(* CoDeSys 2.3 export: TECHMODULE_KINEMATICS.EXP *)
(* Libraries: 03_ApplicationModules\MPLCAxisGroupControl_Kinematics.lib 30.1.17 00:00:00, 03_ApplicationModules\MPLCAxisGroupControl_Kinematics_Internal_Inst1.lib 30.1.17 00:00:00, 04_InterpolatedMotion\MPLCKinematics.lib 30.1.17 00:00:00, 04_InterpolatedMotion\MPLCKinematics_UserKin.lib 30.1.17 00:00:00, 04_InterpolatedMotion\MPLCKinematics_UserLookAhead.lib 30.1.17 00:00:00, 04_InterpolatedMotion\MPLCSimu3D.lib 30.1.17 00:00:00, 11_System\SysLibStr.lib 27.1.17 13:50:06, Internal\MPLCIntern_Kinematics.lib 30.1.17 00:00:00, Internal\MPLCIntern_Kinematics_BC.lib 30.1.17 00:00:00, Internal\MPLCIntern_Kinematics_Small.lib 30.1.17 00:00:00 *)

(* Global variable list: AxisGroupControl_Kinematics/Examples/GlobalVar_AxisGroupControl_Kinematics_Examples *)
VAR_GLOBAL
	(* !!! Do not remove '{flag extrasymbolexport on}'. Otherwise the Kinematics Monitor will not work anymore. *)
	{flag extrasymbolexport on}
	gKinExamples_Control	: ARRAY[1..KIN_AXISGROUPKIN_MAX_NUMBER_OF_KINEMATICS_INSTANCES] OF ST_KinExamples_ControlVariables;
	{flag off}

	gsSeqMode				: ARRAY[1..KIN_AXISGROUPKIN_MAX_NUMBER_OF_KINEMATICS_INSTANCES] OF ST_KinExamples_SequenceType;

	CART_VEL1:ARRAY[1..6] OF LREAL := 1,1,1,1,1,1;  (* VEL 1 [user unit / s] *)
	CART_ACC1:ARRAY[1..6] OF LREAL := 1,1,1,1,1,1;  (*ACC 1 [user unit / (s * s)] *)
	CART_DEC1:ARRAY[1..6] OF LREAL := 1,1,1,1,1,1;  (* DEC 1 [user unit / (s * s)]  *)

	CART_VEL10:ARRAY[1..6] OF LREAL := 10,10,10,10,10,10;  (* VEL 10 [user unit / s] *)
	CART_ACC10:ARRAY[1..6] OF LREAL := 10,10,10,10,10,10;  (*ACC 10 [user unit / (s * s)] *)
	CART_DEC10:ARRAY[1..6] OF LREAL := 10,10,10,10,10,10;  (* DEC 10 [user unit / (s * s)]  *)

	CART_VEL20:ARRAY[1..6] OF LREAL := 20,20,20,20,20,20;  (* VEL 20 [user unit / s] *)
	CART_ACC20:ARRAY[1..6] OF LREAL := 20,20,20,20,20,20;  (*ACC 20 [user unit / (s * s)] *)
	CART_DEC20:ARRAY[1..6] OF LREAL := 20,20,20,20,20,20;  (* DEC 20 [user unit / (s * s)]  *)

	CART_VEL50:ARRAY[1..6] OF LREAL := 50,50,50,50,50,50;  (* VEL 50 [user unit / s] *)
	CART_ACC50:ARRAY[1..6] OF LREAL := 50,50,50,50,50,50;  (*ACC 50 [user unit / (s * s)] *)
	CART_DEC50:ARRAY[1..6] OF LREAL := 50,50,50,50,50,50;  (* DEC 50 [user unit / (s * s)]  *)

	CART_VEL100:ARRAY[1..6] OF LREAL := 100,100,100,100,100,100;  (* VEL 100 [user unit / s] *)
	CART_ACC100:ARRAY[1..6] OF LREAL := 100,100,100,100,100,100;  (*ACC 100 [user unit / (s * s)] *)
	CART_DEC100:ARRAY[1..6] OF LREAL := 100,100,100,100,100,100;  (* DEC 100 [user unit / (s * s)]  *)

	CART_VEL200:ARRAY[1..6] OF LREAL := 200,200,200,200,200,200;  (* VEL 200 [user unit / s] *)
	CART_ACC200:ARRAY[1..6] OF LREAL := 200,200,200,200,200,200;  (*ACC 200 [user unit / (s * s)] *)
	CART_DEC200:ARRAY[1..6] OF LREAL := 200,200,200,200,200,200;  (* DEC 200 [user unit / (s * s)]  *)

	CART_VEL1000:ARRAY[1..6] OF LREAL := 1000,1000,1000,1000,1000,1000;  (* VEL 1000 [user unit / s] *)
	CART_ACC1000:ARRAY[1..6] OF LREAL := 1000,1000,1000,1000,1000,1000;  (*ACC 1000 [user unit / (s * s)] *)
	CART_DEC1000:ARRAY[1..6] OF LREAL := 1000,1000,1000,1000,1000,1000;  (* DEC 1000 [user unit / (s * s)]  *)

	CART_JERK100:ARRAY[1..6] OF LREAL := 100,100,100,100,100,100;  (* JERK  [ms] *)

	AXIS_VEL100:ARRAY[1..8] OF LREAL := 100,100,100,100,100,100,100,100;  (* VEL 100 [user unit / s] *)
	AXIS_ACC100:ARRAY[1..8] OF LREAL := 100,100,100,100,100,100,100,100;  (*ACC 100 [user unit / (s * s)] *)
	AXIS_DEC100:ARRAY[1..8] OF LREAL := 100,100,100,100,100,100,100,100;  (* DEC 100 [user unit / (s * s)]  *)
	AXIS_JERK100:ARRAY[1..8] OF LREAL := 100,100,100,100,100,100,100,100;  (* JERK  [ms] *)

	KIN_NO_SYNC: ARRAY[0..8]OF BOOL := FALSE, FALSE, FALSE, FALSE, FALSE, FALSE, FALSE, FALSE, FALSE;

(* PRG_XYZ_FillQueue_LIN3D_with_Array *)
	points: ARRAY[1..10] OF ST_AxisGroupKin_Point;
(* PRG_XYZ_USER poses and parameters *)
	XYZ_USER_P1 : ARRAY[1..8] OF LREAL := 10,10,0;
	XYZ_USER_P2 : ARRAY[1..8] OF LREAL := 200,200,200;
(* PRG_XYZ_PICKnPLACE poses and parameters *)
	XYZ_PICKnPLACE_P1 : ARRAY[1..8] OF LREAL := 10,0,0;
	XYZ_PICKnPLACE_P2 : ARRAY[1..8] OF LREAL := 10,0,200;
	XYZ_PICKnPLACE_P3 : ARRAY[1..8] OF LREAL := 300,0,200;
	XYZ_PICKnPLACE_P4 : ARRAY[1..8] OF LREAL := 300,0,0;
	XYZ_PICKnPLACE_BlendingDistance : LREAL := 50;
(* PRG_XYZ_LIN_CIRC_LIN poses and parameters *)
	XYZ_TARG_LIN_CIRC_P1 : ARRAY[1..8] OF LREAL := 10,10,0;
	XYZ_TARG_LIN_CIRC_P2 : ARRAY[1..8] OF LREAL := 100,10,0;
	XYZ_TARG_LIN_CIRC_R3 : LREAL := 50;
	XYZ_TARG_LIN_CIRC_A3 : LREAL := 180;
	XYZ_TARG_LIN_CIRC_P4 : ARRAY[1..8] OF LREAL := 10,200,0;

END_VAR

(* Global variable list: AxisGroupControl_Kinematics/GlobalVar_AxisGroupControl_Kinematics *)
VAR_GLOBAL
	{flag extrasymbolexport on}
	AxisGroupKin 		: ST_AxisGroupKin;
	{flag off}
END_VAR

(* Global variable list: AxisGroupControl_Kinematics/Version_AxisGroupControl_Kinematics *)
VAR_GLOBAL
	VERSION_AXISGROUPCONTROL_KINEMATICS : DWORD := 180;
	RELEASE_AXISGROUPCONTROL_KINEMATICS : DWORD := 100;
END_VAR

(* Data type in AxisGroupControl_Kinematics/Examples *)
TYPE ENUM_AxisIndex :(
	A1:=1,
	A2:=2,
	A3:=3,
	A4:=4,
	A5:=5,
	A6:=6,
	A7:=7,
	A8:=8
);
END_TYPE

(* Data type in AxisGroupControl_Kinematics/Examples *)
TYPE ENUM_CartIndex :(
	X:=1,
	Y:=2,
	Z:=3,
	A:=4,
	B:=5,
	C:=6


);
END_TYPE

(* Data type in AxisGroupControl_Kinematics/Examples *)
TYPE ST_AxisGroupKin_Point :
STRUCT
	x: LREAL;
	y: LREAL;
	z: LREAL;
	A: LREAL;
	B: LREAL;
	C: LREAL;
END_STRUCT
END_TYPE

(* Data type in AxisGroupControl_Kinematics/Examples *)
TYPE ST_KinExamples_ControlVariables :
STRUCT
	EnableExamples		: BOOL;

	ProgramNumber 		: DINT := 1;
	ErrorReset 			: BOOL;

	Kin 					: ST_KinExamples_ControlVariables_Kin;
	Inverter				: ST_KinExamples_ControlVariables_Inverter;


END_STRUCT
END_TYPE

(* Data type in AxisGroupControl_Kinematics/Examples *)
TYPE ST_KinExamples_ControlVariables_Inverter :
STRUCT

	Enable_Stop_AllAxis			: BOOL;
	Enable_RapidStop_AllAxis	: BOOL;
	Inhibit_AllAxis 					: BOOL;

END_STRUCT
END_TYPE

(* Data type in AxisGroupControl_Kinematics/Examples *)
TYPE ST_KinExamples_ControlVariables_Kin :
STRUCT

	FeedEnable 			: BOOL;
	RapidStop 			: BOOL;
	OverridePercentage 	: INT := 10;

END_STRUCT
END_TYPE

(* Data type in AxisGroupControl_Kinematics/Examples *)
TYPE ST_KinExamples_SequenceType :
STRUCT
	Reset: BOOL;						(*Die Variable verhält sich ähnlich wie SFCInit. Im Unterschied zu dieser wird allerdings nach der Initialisierungder Init-Schritt weiter abgearbeitet.
										So könnte beispielsweise im Init-Schritt das Flag SFCReset gleich wieder auf FALSE gesetzt werden.*)
	Init: BOOL;							(*Wenn die Variable TRUE ist, wird die Ablaufsprache auf den Init-Schritt zurückgesetzt.
										Die anderen AS-Flags werden ebenfalls zurückgesetzt (Initialisierung). 
										Solange die Variable TRUE ist, bleibt der Init-Schritt gesetzt (aktiv), wird aber nicht ausgeführt.
										Erst wenn SFCInit wieder auf FALSE gesetzt wird, wird der Baustein normal weiterbearbeitet.*)
	EnableLimit: BOOL;				(*Wenn die Variable TRUE ist, werden Zeitüberschreitungen bei den Schritten in SFCError registriert.
										Ansonsten werden Zeitüberschreitungen ignoriert.
										Das Flag kann beispielsweise bei Inbetriebnahme oder Handbetrieb nützlich sein.*)
	QuitError: BOOL;					(*Solange die Variable TRUE ist, wird die Abarbeitung des AS-Diagramms angehalten.
										Eine in der Variablen SFCError registrierte Zeitüberschreitung wird dabei zurückgesetzt. 
										Wenn die Variable wieder auf FALSE gesetzt wird, werden alle bisherigen Zeiten in den aktiven Schritten zurückgesetzt.
										Voraussetzung dafür ist die Deklaration der Variablen SFCError, die die Zeitüberschreitung registriert.*)
	CurrentStep: STRING;			(*In dieser Variablen wird der Name des momentan akitven Schritts gespeichert, unabhängig von der Zeitüberwachung.
										Bei einer Paralellverzweigung wird der Name des Schritts im äußersten rechten Zweig gespeichert*)
	Error: BOOL;						(*Diese Variable wird TRUE, wenn in einem AS-Diagramm eine Zeitüberschreitung aufgetreten ist.
										Wenn nach der ersten Zeitüberschreitung eine weitere auftritt, wird diese nicht mehr registriert, 
										es sei denn, die Variable SFCError wurde vorher wieder zurückgesetzt. 
										Die Deklaration von SFCError ist Voraussetzung für das Funktionieren der anderen Flag-Variablen,
										die zur Kontrolle des zeitlichen Ablaufs dienen (SFCErrorStep, SFCErrorPOU, SFCQuitError, SFCErrorAnalyzationTable.*)
	ErrorStep: STRING; 				(*Wenn in SFCError eine Zeitüberschreitung im AS-Diagramm registriert wird, speichert die Variable den Namen des Schritts,
										der die Zeitüberschreitung verursacht hat.
										Voraussetzung dafür ist die Deklaration der Variablen SFCError, die die Zeitüberschreitung registriert. *)
	Done: BOOL;
END_STRUCT
END_TYPE

(* POU AxisGroupControl_Kinematics/Examples/Simu3D_Show User Positions/PRG_UserCoordSystems_Example, ST *)
(*##############################################################################################################

	IMPORTANT NOTICE:
 	This example is a special and free service that demonstrates only the basic 
	approach to generating a PLC program as a non-binding sample. 
	SEW is not liable for the contents of the sample program.

	Name:			PRG_Example_UserCoordSystems
	Job:			This example shows, how you can display user defined positions in the 3D Simulation. They are shown as coordinate systems. 

					The struct 'Example_CoordSystems' contains the data for the visualization.
					With the variables 'Example_CoordSystems.CS[1].WCS_XCS[1..6]' you can change the postition of the coordinate systems.
					In the action 'Configuration' you can change the amount of coordinate systems ('Example_CoordSystems.Config.NumberOfCoordSystems') and the names/labels that are displayed in the 3D Simulation.

					Call this Programm in the TaskLowPriority.	

################################################################################################################*)
PROGRAM PRG_UserCoordSystems_Example
VAR

	Example_CoordSystems						 : ST_Simu3D_CoordSystems;	(* Datastructure/Interface for the coordinate systems *)
	fbFB_Simu3D_DataExchange_CoordSys 	 :  FB_Simu3D_DataExchange_CoordSys;	(* This FB manages the communication with the PC/simulation tool *)
	bCoordSystemsConfigured	: BOOL:=FALSE;
	iCoordSysCounter : INT;

END_VAR
IF NOT bCoordSystemsConfigured THEN
	Configuration();
ELSE
	Example_CoordSystems.EnableVisu := TRUE; (* Start the communication with the PC after the configuration is done *)

	Example_CoordSystems.CS[1].WCS_XCS[1] := 50; (* example for changing the position (here only x coordinate) of the first coordinate system *)

	fbFB_Simu3D_DataExchange_CoordSys(CoordSystems := Example_CoordSystems);
END_IF
END_PROGRAM
ACTION Configuration:
IF AxisGroupKin.ConfigDataAvailable THEN

	Example_CoordSystems.Config.Simu3D_Config.Content1_FileName := ''; (* Do not change. *)
	Example_CoordSystems.Config.Simu3D_Config.Content1_Coding := 138; (* Do not change. *)
	Example_CoordSystems.Config.Simu3D_Config.Content2_Coding := 84; (* Do not change. *)
	Example_CoordSystems.Config.Simu3D_Config.Content2_FileName := 'UserCoordsystems.csb'; (* Do not change. *)
	Example_CoordSystems.Config.Simu3D_Config.WriteDiagToMemoryCard := FALSE; (* Do not change. *)
	Example_CoordSystems.Config.Simu3D_Config.KeepSceneAtLoading := TRUE; (* Do not change. *)

	Example_CoordSystems.Config.strInstanceName := 'Example_UserCoordsystems'; (* Name of the group of coordinate systems which is displayed at bottom left of 3D simulation *)
	Example_CoordSystems.Config.NumberOfCoordSystems := 1; (* Determines how many coordinate systems are display. Maximum amount of coordinate systems  is NUM_OF_USER_COORDSYSTEMS_PER_INSTANCE (= 20) *)

	(* Use the IP-Address and RotUnit of the first Kinematics-Instance *)
	Example_CoordSystems.Config.Simu3D_Config.IP_Address_PC := AxisGroupKin.Inst[1].Config.Simu3D.IP_Address_SimulationPC;
	IF AxisGroupKin.Inst[1].Config.Cart.Use[4] = KIN_USE_DEGR THEN
		Example_CoordSystems.Config.UseDegree := TRUE;
	ELSE
		Example_CoordSystems.Config.UseDegree := FALSE;
	END_IF

	FOR iCoordSysCounter := 1 TO Example_CoordSystems.Config.NumberOfCoordSystems DO
		Example_CoordSystems.CS[iCoordSysCounter].Label := CONCAT('Example_P', INT_TO_STRING(iCoordSysCounter)); (* text displayed at each coordinate sytem *)
	END_FOR

	bCoordSystemsConfigured := TRUE;

END_IF
END_ACTION

(* POU PRG_Kinematics/PRG_TaskMain_Kinematics, ST *)
PROGRAM PRG_TaskMain_Kinematics
VAR
	fbUser_Kinematics_Examples : ARRAY[1..KIN_AXISGROUPKIN_MAX_NUMBER_OF_KINEMATICS_INSTANCES] OF FB_User_Kinematics_Examples;
	i : INT;
END_VAR
(*#######################################################################################

	PRG_TaskMain_Kinematics

	ToDo: Call this program in the task configuration after PRG_TaskMain();

#########################################################################################*)

(* Examples for common motion sequences *)
FOR i := 1 TO KIN_AXISGROUPKIN_MAX_NUMBER_OF_KINEMATICS_INSTANCES DO
	fbUser_Kinematics_Examples[i](AxisGroupKin_Inst := AxisGroupKin.Inst[i]);
END_FOR

(* Do not remove! *)
AxisGroupControl_Configuration_Kinematics(Enable := TRUE);

(* Do not remove! *)
AxisGroupControl_Main_Kinematics(Enable := TRUE);
END_PROGRAM

(* POU AxisGroupControl_Kinematics/Examples/FB_User_Kinematics_Examples, FBD *)
(*##############################################################################################################

	IMPORTANT NOTICE:
 	This example is a special and free service that demonstrates only the basic 
	approach to generating a PLC program as a non-binding sample. 
	SEW is not liable for the contents of the sample program.

	Name:			FB_User_Kinematics_Examples
	Job:			This FB is called in  PRG_TaskMain_Kinematics and calls all the User programs

################################################################################################################*)

FUNCTION_BLOCK FB_User_Kinematics_Examples
VAR
	fbMainCycle_Kinematics	: MainCycle_Kinematics;
	F_TRIG: F_TRIG;

END_VAR
VAR_IN_OUT
	AxisGroupKin_Inst : ST_AxisGroupKin_Instance;				(* AxisGroupControl Interface to application program *)
END_VAR
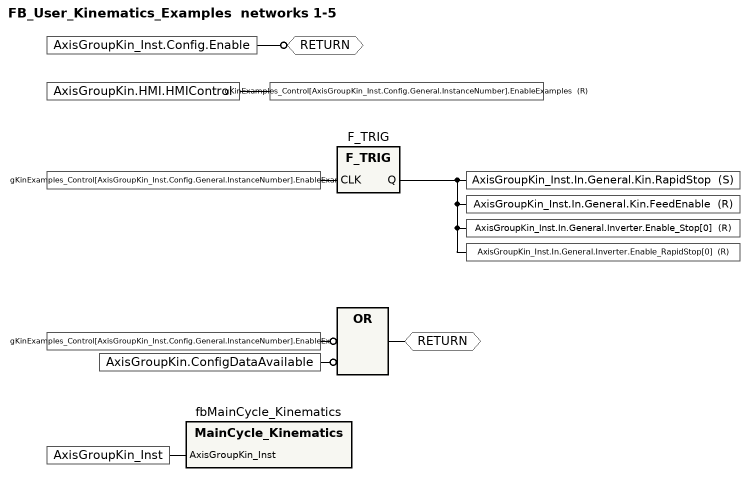
_FBD_ (* Function Block Diagram *)
NETWORK 1 (* Don't run the example programs, if the kinematics instance is not enabled. *)
	NOT AxisGroupKin_Inst.Config.Enable => <RETURN>
NETWORK 2 (* If the HMIControl is True the UserProgramm must not be executed, because otherwise the KinematicsMonitor has no control over the AxisGroupKin Interface *)
	AxisGroupKin.HMI.HMIControl => R gKinExamples_Control[AxisGroupKin_Inst.Config.General.InstanceNumber].EnableExamples
NETWORK 3 (* At reset of EnableExamples, stop the motion. *)
	F_TRIG:F_TRIG(CLK: gKinExamples_Control[AxisGroupKin_Inst.Config.General.InstanceNumber].EnableExamples) => S AxisGroupKin_Inst.In.General.Kin.RapidStop, R AxisGroupKin_Inst.In.General.Kin.FeedEnable, R AxisGroupKin_Inst.In.General.Inverter.Enable_Stop[0], R AxisGroupKin_Inst.In.General.Inverter.Enable_RapidStop[0]
NETWORK 4 (* Don't execute any motion sequence before AxisGroupKin.ConfigDataAvailable = TRUE. *)
	OR(NOT gKinExamples_Control[AxisGroupKin_Inst.Config.General.InstanceNumber].EnableExamples, NOT AxisGroupKin.ConfigDataAvailable) => <RETURN>
NETWORK 5
	fbMainCycle_Kinematics:MainCycle_Kinematics(AxisGroupKin_Inst: AxisGroupKin_Inst)
_END_FBD_
(* the same logic as Structured Text *)
(* Network 1: Don't run the example programs, if the kinematics instance is not enabled. *)
IF NOT AxisGroupKin_Inst.Config.Enable THEN RETURN; END_IF;
(* Network 2: If the HMIControl is True the UserProgramm must not be executed, because otherwise the KinematicsMonitor has no control over the AxisGroupKin Interface *)
IF AxisGroupKin.HMI.HMIControl THEN gKinExamples_Control[AxisGroupKin_Inst.Config.General.InstanceNumber].EnableExamples := FALSE; END_IF;
(* Network 3: At reset of EnableExamples, stop the motion. *)
F_TRIG(CLK := gKinExamples_Control[AxisGroupKin_Inst.Config.General.InstanceNumber].EnableExamples);
IF F_TRIG.Q THEN AxisGroupKin_Inst.In.General.Kin.RapidStop := TRUE; AxisGroupKin_Inst.In.General.Kin.FeedEnable := FALSE; AxisGroupKin_Inst.In.General.Inverter.Enable_Stop[0] := FALSE; AxisGroupKin_Inst.In.General.Inverter.Enable_RapidStop[0] := FALSE; END_IF;
(* Network 4: Don't execute any motion sequence before AxisGroupKin.ConfigDataAvailable = TRUE. *)
IF NOT gKinExamples_Control[AxisGroupKin_Inst.Config.General.InstanceNumber].EnableExamples OR NOT AxisGroupKin.ConfigDataAvailable THEN RETURN; END_IF;
(* Network 5 *)
fbMainCycle_Kinematics(AxisGroupKin_Inst := AxisGroupKin_Inst);
END_FUNCTION_BLOCK

(* POU AxisGroupControl_Kinematics/Examples/MainCycle_Kinematics, SFC *)
(*##############################################################################################################

	IMPORTANT NOTICE:
 	This example is a special and free service that demonstrates only the basic 
	approach to generating a PLC program as a non-binding sample. 
	SEW is not liable for the contents of the sample program.

	Name:			MainCycle_MDX
	Job:			Calls all UserProgramms

################################################################################################################*)
FUNCTION_BLOCK MainCycle_Kinematics
VAR_INPUT
END_VAR
VAR_OUTPUT
END_VAR
VAR
	fbOperationMode			: OperationMode_Kinematics;
	InstanceNumber				: INT;
	i : INT;
END_VAR
VAR_IN_OUT
	AxisGroupKin_Inst : ST_AxisGroupKin_Instance;				(* AxisGroupControl Interface to application program *)
END_VAR
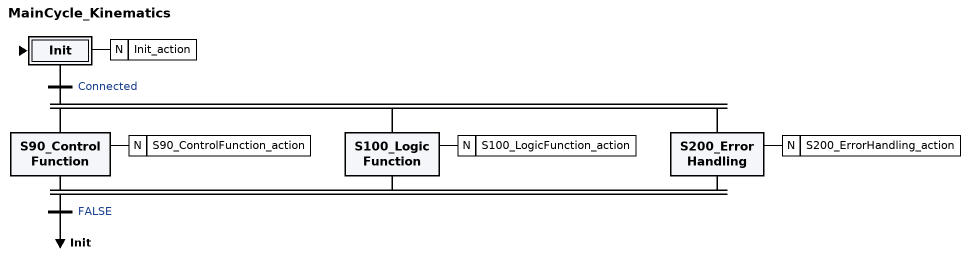
INITIAL_STEP Init:
	Init_action(N);
END_STEP
TRANSITION FROM Init TO (S90_ControlFunction, S100_LogicFunction, S200_ErrorHandling) := Connected;
END_TRANSITION
STEP S90_ControlFunction:
	S90_ControlFunction_action(N);
END_STEP
STEP S100_LogicFunction:
	S100_LogicFunction_action(N);
END_STEP
STEP S200_ErrorHandling:
	S200_ErrorHandling_action(N);
END_STEP
TRANSITION FROM (S90_ControlFunction, S100_LogicFunction, S200_ErrorHandling) TO Init := FALSE;
END_TRANSITION

ACTION Init_action:
InstanceNumber := AxisGroupKin_Inst.Config.General.InstanceNumber;

FOR i := 1 TO 8 DO
	AxisGroupKin_Inst.In.General.Inverter.Enable_RapidStop[i] := FALSE;
	AxisGroupKin_Inst.In.General.Inverter.Enable_Stop[i] := FALSE;
	AxisGroupKin_Inst.In.General.Inverter.Inhibit[i] := FALSE;
END_FOR
END_ACTION

ACTION S90_ControlFunction_action:
AxisGroupKin_Inst.In.General.Inverter.Enable_RapidStop[0]	:= gKinExamples_Control[InstanceNumber].Inverter.Enable_RapidStop_AllAxis;
AxisGroupKin_Inst.In.General.Inverter.Enable_Stop[0] 			:= gKinExamples_Control[InstanceNumber].Inverter.Enable_Stop_AllAxis;
AxisGroupKin_Inst.In.General.Inverter.Inhibit[0]					:= gKinExamples_Control[InstanceNumber].Inverter.Inhibit_AllAxis;

AxisGroupKin_Inst.In.General.Kin.FeedEnable					:= gKinExamples_Control[InstanceNumber].Kin.FeedEnable;
AxisGroupKin_Inst.In.General.Kin.RapidStop					:= gKinExamples_Control[InstanceNumber].Kin.RapidStop;
AxisGroupKin_Inst.In.General.Kin.OverridePercentage			:= gKinExamples_Control[InstanceNumber].Kin.OverridePercentage;

AxisGroupKin_Inst.In.General.Reset 							:= gKinExamples_Control[InstanceNumber].ErrorReset;
END_ACTION

ACTION S100_LogicFunction_action:
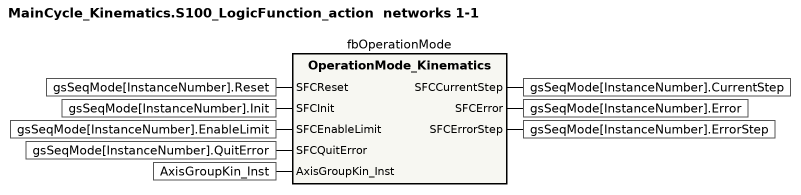
_FBD_ (* Function Block Diagram *)
NETWORK 1 (* In the FB Operation Mode the switch on sequense and running the Sequence Programms is implemented. *)
	fbOperationMode:OperationMode_Kinematics(SFCReset: gsSeqMode[InstanceNumber].Reset, SFCInit: gsSeqMode[InstanceNumber].Init, SFCEnableLimit: gsSeqMode[InstanceNumber].EnableLimit, SFCQuitError: gsSeqMode[InstanceNumber].QuitError, AxisGroupKin_Inst: AxisGroupKin_Inst, SFCError => gsSeqMode[InstanceNumber].Error, SFCErrorStep => gsSeqMode[InstanceNumber].ErrorStep) => gsSeqMode[InstanceNumber].CurrentStep
_END_FBD_
(* the same logic as Structured Text *)
(* Network 1: In the FB Operation Mode the switch on sequense and running the Sequence Programms is implemented. *)
fbOperationMode(SFCReset := gsSeqMode[InstanceNumber].Reset, SFCInit := gsSeqMode[InstanceNumber].Init, SFCEnableLimit := gsSeqMode[InstanceNumber].EnableLimit, SFCQuitError := gsSeqMode[InstanceNumber].QuitError, AxisGroupKin_Inst := AxisGroupKin_Inst);
gsSeqMode[InstanceNumber].Error := fbOperationMode.SFCError;
gsSeqMode[InstanceNumber].ErrorStep := fbOperationMode.SFCErrorStep;
gsSeqMode[InstanceNumber].CurrentStep := fbOperationMode.SFCCurrentStep;
END_ACTION

ACTION S200_ErrorHandling_action:
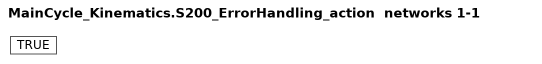
_FBD_ (* Function Block Diagram *)
NETWORK 1
	TRUE
_END_FBD_
(* the same logic as Structured Text *)
(* Network 1 *)
END_ACTION

TRANSITION Connected:
_FBD_ (* Function Block Diagram *)
NETWORK 1
	AxisGroupKin.Inst[InstanceNumber].Out.General.Inverter.Connected[0]
_END_FBD_
(* the same logic as Structured Text *)
(* Network 1 *)
Connected := AxisGroupKin.Inst[InstanceNumber].Out.General.Inverter.Connected[0];
END_TRANSITION
END_FUNCTION_BLOCK

(* POU AxisGroupControl_Kinematics/Examples/OperationMode_Kinematics, SFC *)
(*##############################################################################################################

	IMPORTANT NOTICE:
 	This example is a special and free service that demonstrates only the basic 
	approach to generating a PLC program as a non-binding sample. 
	SEW is not liable for the contents of the sample program.

	Name:			OperationMode
	Job:			Calls all kinematics example programs

################################################################################################################*)
FUNCTION_BLOCK OperationMode_Kinematics
VAR_INPUT
	SFCReset:						 BOOL;									(*This variable, of type BOOL, behaves similarly to SFCInit. Unlike the latter, however,
																				further processing takes place after the initialization of the Init step.
																				Thus for example the SFCReset flag could be re-set to FALSE in the Init step.*)

	SFCInit:							 BOOL;									(*When this boolean variable has the value TRUE the sequential function chart is set back
																				to the Init step. The other SFC flags are reset too (initialization).
																				The Init step remains active, but is not executed, for as long as the variable has the value TRUE.
																				It is only when SFCInit is again set to FALSE that the block can be processed normally.*)
	SFCEnableLimit:					BOOL;									(*This variable is of the type BOOL. When it has the value TRUE, the timeouts of the
																				steps will be registered in SFCError. Other timeouts will be ignored.*)
	SFCQuitError: 						BOOL;									(*Provided that the Execution of the SFC diagram is stopped for as long as this boolean
																				variable has the value TRUE whereby a possible timeout in the variable SFCError is reset. All
																				previous times in the active steps are reset when the variable again assumes the value FALSE. It is a
																				pre-condition that the flag SFCError has been defined also, which registers any timeout in the SFC.*)
END_VAR
VAR_OUTPUT
	SFCCurrentStep:					 STRING;								(*This variable is of the type STRING.
																				The name of the step is stored in this variable which is active, independently of the time monitoring.
																				In the case of simultaneous sequences the step is stored in the branch on the outer right.*)
	SFCError: 							BOOL;									(*This Boolean variable is TRUE when a timeout has occurred in a SFC diagram. If another
																				timeout occurs in a program after the first one, it will not be registered unless the variable SFCError is
																				reset first. It is a pre-condition that SFCError is defined, if you want to use the other time-controlling
																				flags (SFCErrorStep, SFCErrorPOU, SFCQuitError, SFCErrorAnalyzation).*)
	SFCErrorStep: 					STRING; 								(*This variable is of the type STRING. If SFCError registers a timeout, in this variable is
																				stored the name of the step which has caused the timeout. It is a pre-condition that the flag SFCError
																				has been defined also, which registers any timeout in the SFC. *)
END_VAR
VAR_IN_OUT
	AxisGroupKin_Inst				: ST_AxisGroupKin_Instance;				(* AxisGroupControl Interface to application program *)
END_VAR
VAR
	fbPRG_XYZ_PICKnPLACE_ST							: PRG01_XYZ_PICKnPLACE_ST;
	fbPRG_XYZ_PICKnPLACE_SFC							: PRG02_XYZ_PICKnPLACE_SFC;
	fbPRG_XYZ_TARG_LIN_CIRC_ST						: PRG03_XYZ_TARG_LIN_CIRC_ST;
	fbPRG_XYZ_TARG_LIN_CIRC_SFC						: PRG04_XYZ_TARG_LIN_CIRC_SFC;
	fbPRG_XYZ_FillQueue_LIN3D_with_Array_ST			: PRG05_XYZ_FillQueue_LIN3D_with_Array_ST;
	fbPRG_XYZ_FillQueue_LIN3D_with_Array_SFC		: PRG06_XYZ_FillQueue_LIN3D_with_Array_SFC;
	fbPRG_XYZ_USER_ST									: PRG07_XYZ_USER_ST;
	fbPRG_XYZ_USER_SFC									: PRG08_XYZ_USER_SFC;
	InstanceNumber: INT;
END_VAR
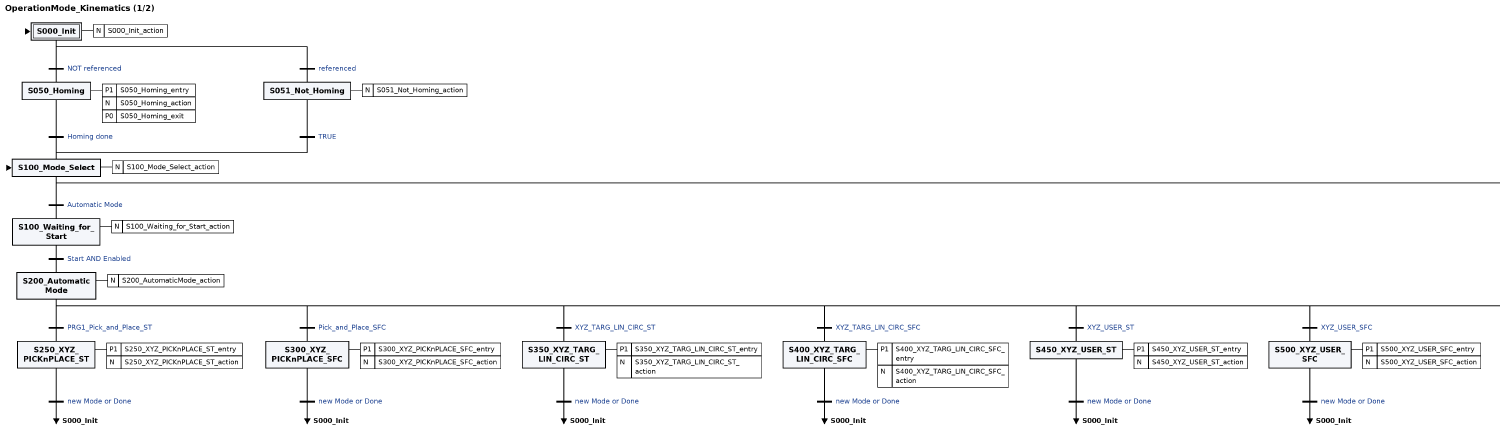
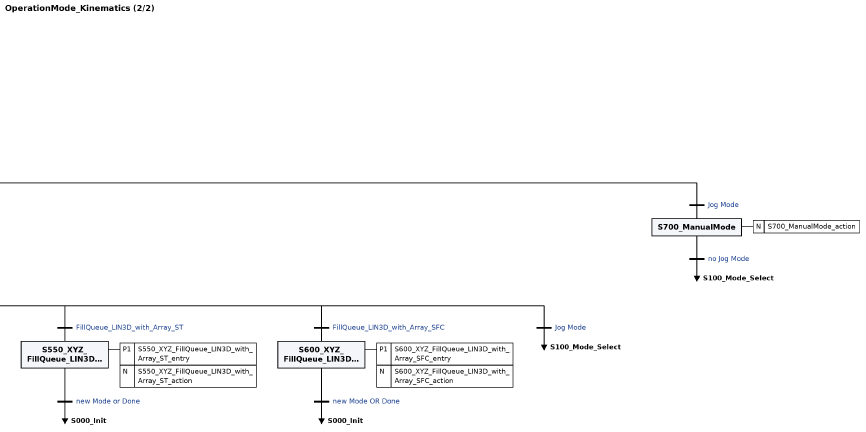
INITIAL_STEP S000_Init:
	S000_Init_action(N);
END_STEP
TRANSITION FROM S000_Init TO S050_Homing := NOT referenced;
END_TRANSITION
TRANSITION FROM S000_Init TO S051_Not_Homing := referenced;
END_TRANSITION
STEP S051_Not_Homing:
	S051_Not_Homing_action(N);
END_STEP
TRANSITION FROM S051_Not_Homing TO S100_Mode_Select := TRUE;
END_TRANSITION
STEP S050_Homing:
	S050_Homing_entry(P1);
	S050_Homing_action(N);
	S050_Homing_exit(P0);
END_STEP
TRANSITION FROM S050_Homing TO S100_Mode_Select := Homing done;
END_TRANSITION
STEP S100_Mode_Select:
	S100_Mode_Select_action(N);
END_STEP
TRANSITION FROM S100_Mode_Select TO S100_Waiting_for_Start := Automatic Mode;
END_TRANSITION
TRANSITION FROM S100_Mode_Select TO S700_ManualMode := Jog Mode;
END_TRANSITION
STEP S700_ManualMode:
	S700_ManualMode_action(N);
END_STEP
TRANSITION FROM S700_ManualMode TO S100_Mode_Select := no Jog Mode;
END_TRANSITION
STEP S100_Waiting_for_Start:
	S100_Waiting_for_Start_action(N);
END_STEP
TRANSITION FROM S100_Waiting_for_Start TO S200_AutomaticMode := Start AND Enabled;
END_TRANSITION
STEP S200_AutomaticMode:
	S200_AutomaticMode_action(N);
END_STEP
TRANSITION FROM S200_AutomaticMode TO S250_XYZ_PICKnPLACE_ST := PRG1_Pick_and_Place_ST;
END_TRANSITION
TRANSITION FROM S200_AutomaticMode TO S300_XYZ_PICKnPLACE_SFC := Pick_and_Place_SFC;
END_TRANSITION
TRANSITION FROM S200_AutomaticMode TO S350_XYZ_TARG_LIN_CIRC_ST := XYZ_TARG_LIN_CIRC_ST;
END_TRANSITION
TRANSITION FROM S200_AutomaticMode TO S400_XYZ_TARG_LIN_CIRC_SFC := XYZ_TARG_LIN_CIRC_SFC;
END_TRANSITION
TRANSITION FROM S200_AutomaticMode TO S450_XYZ_USER_ST := XYZ_USER_ST;
END_TRANSITION
TRANSITION FROM S200_AutomaticMode TO S500_XYZ_USER_SFC := XYZ_USER_SFC;
END_TRANSITION
TRANSITION FROM S200_AutomaticMode TO S550_XYZ_FillQueue_LIN3D_with_Array_ST := FillQueue_LIN3D_with_Array_ST;
END_TRANSITION
TRANSITION FROM S200_AutomaticMode TO S600_XYZ_FillQueue_LIN3D_with_Array_SFC := FillQueue_LIN3D_with_Array_SFC;
END_TRANSITION
TRANSITION FROM S200_AutomaticMode TO S100_Mode_Select := Jog Mode;
END_TRANSITION
STEP S300_XYZ_PICKnPLACE_SFC:
	S300_XYZ_PICKnPLACE_SFC_entry(P1);
	S300_XYZ_PICKnPLACE_SFC_action(N);
END_STEP
TRANSITION FROM S300_XYZ_PICKnPLACE_SFC TO S000_Init := new Mode or Done;
END_TRANSITION
STEP S350_XYZ_TARG_LIN_CIRC_ST:
	S350_XYZ_TARG_LIN_CIRC_ST_entry(P1);
	S350_XYZ_TARG_LIN_CIRC_ST_action(N);
END_STEP
TRANSITION FROM S350_XYZ_TARG_LIN_CIRC_ST TO S000_Init := new Mode or Done;
END_TRANSITION
STEP S400_XYZ_TARG_LIN_CIRC_SFC:
	S400_XYZ_TARG_LIN_CIRC_SFC_entry(P1);
	S400_XYZ_TARG_LIN_CIRC_SFC_action(N);
END_STEP
TRANSITION FROM S400_XYZ_TARG_LIN_CIRC_SFC TO S000_Init := new Mode or Done;
END_TRANSITION
STEP S450_XYZ_USER_ST:
	S450_XYZ_USER_ST_entry(P1);
	S450_XYZ_USER_ST_action(N);
END_STEP
TRANSITION FROM S450_XYZ_USER_ST TO S000_Init := new Mode or Done;
END_TRANSITION
STEP S500_XYZ_USER_SFC:
	S500_XYZ_USER_SFC_entry(P1);
	S500_XYZ_USER_SFC_action(N);
END_STEP
TRANSITION FROM S500_XYZ_USER_SFC TO S000_Init := new Mode or Done;
END_TRANSITION
STEP S550_XYZ_FillQueue_LIN3D_with_Array_ST:
	S550_XYZ_FillQueue_LIN3D_with_Array_ST_entry(P1);
	S550_XYZ_FillQueue_LIN3D_with_Array_ST_action(N);
END_STEP
TRANSITION FROM S550_XYZ_FillQueue_LIN3D_with_Array_ST TO S000_Init := new Mode or Done;
END_TRANSITION
STEP S600_XYZ_FillQueue_LIN3D_with_Array_SFC:
	S600_XYZ_FillQueue_LIN3D_with_Array_SFC_entry(P1);
	S600_XYZ_FillQueue_LIN3D_with_Array_SFC_action(N);
END_STEP
TRANSITION FROM S600_XYZ_FillQueue_LIN3D_with_Array_SFC TO S000_Init := new Mode OR Done;
END_TRANSITION
STEP S250_XYZ_PICKnPLACE_ST:
	S250_XYZ_PICKnPLACE_ST_entry(P1);
	S250_XYZ_PICKnPLACE_ST_action(N);
END_STEP
TRANSITION FROM S250_XYZ_PICKnPLACE_ST TO S000_Init := new Mode or Done;
END_TRANSITION

ACTION S000_Init_action:
InstanceNumber							:= AxisGroupKin_Inst.Config.General.InstanceNumber;
gsSeqMode[InstanceNumber].Reset	:= FALSE;
END_ACTION

ACTION S051_Not_Homing_action:
_FBD_ (* Function Block Diagram *)
_END_FBD_
END_ACTION

ACTION S050_Homing_entry:
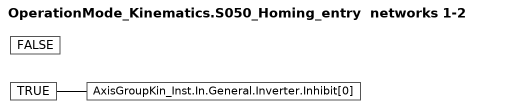
_FBD_ (* Function Block Diagram *)
NETWORK 1 (* Entry Action for Homing *)
	FALSE
NETWORK 2
	TRUE => AxisGroupKin_Inst.In.General.Inverter.Inhibit[0]
_END_FBD_
(* the same logic as Structured Text *)
(* Network 1: Entry Action for Homing *)
(* Network 2 *)
AxisGroupKin_Inst.In.General.Inverter.Inhibit[0] := TRUE;
END_ACTION

ACTION S050_Homing_action:
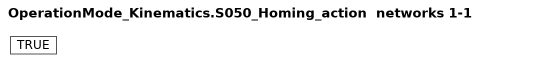
_FBD_ (* Function Block Diagram *)
NETWORK 1 (* Action for Homing *)
	TRUE
_END_FBD_
(* the same logic as Structured Text *)
(* Network 1: Action for Homing *)
END_ACTION

ACTION S050_Homing_exit:
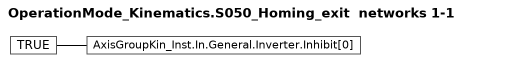
_FBD_ (* Function Block Diagram *)
NETWORK 1
	TRUE => AxisGroupKin_Inst.In.General.Inverter.Inhibit[0]
_END_FBD_
(* the same logic as Structured Text *)
(* Network 1 *)
AxisGroupKin_Inst.In.General.Inverter.Inhibit[0] := TRUE;
END_ACTION

ACTION S100_Mode_Select_action:
(* @TEXT_IMPLEMENTATION := 'ST' *)
AxisGroupKin_Inst.In.General.Mode:=KIN_STOP;
END_ACTION

ACTION S700_ManualMode_action:
(* @TEXT_IMPLEMENTATION := 'ST' *)
;
END_ACTION

ACTION S100_Waiting_for_Start_action:
(* @TEXT_IMPLEMENTATION := 'ST' *)
;
END_ACTION

ACTION S200_AutomaticMode_action:
_FBD_ (* Function Block Diagram *)
_END_FBD_
END_ACTION

ACTION S300_XYZ_PICKnPLACE_SFC_entry:
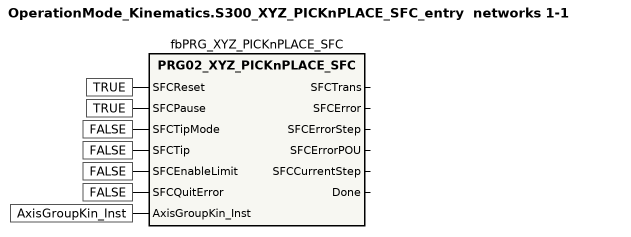
_FBD_ (* Function Block Diagram *)
NETWORK 1
	fbPRG_XYZ_PICKnPLACE_SFC:PRG02_XYZ_PICKnPLACE_SFC(SFCReset: TRUE, SFCPause: TRUE, SFCTipMode: FALSE, SFCTip: FALSE, SFCEnableLimit: FALSE, SFCQuitError: FALSE, AxisGroupKin_Inst: AxisGroupKin_Inst)
_END_FBD_
(* the same logic as Structured Text *)
(* Network 1 *)
fbPRG_XYZ_PICKnPLACE_SFC(SFCReset := TRUE, SFCPause := TRUE, SFCTipMode := FALSE, SFCTip := FALSE, SFCEnableLimit := FALSE, SFCQuitError := FALSE, AxisGroupKin_Inst := AxisGroupKin_Inst);
END_ACTION

ACTION S300_XYZ_PICKnPLACE_SFC_action:
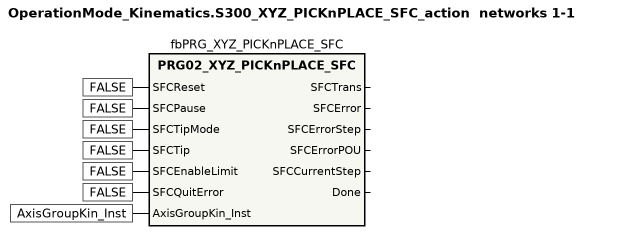
_FBD_ (* Function Block Diagram *)
NETWORK 1
	fbPRG_XYZ_PICKnPLACE_SFC:PRG02_XYZ_PICKnPLACE_SFC(SFCReset: FALSE, SFCPause: FALSE, SFCTipMode: FALSE, SFCTip: FALSE, SFCEnableLimit: FALSE, SFCQuitError: FALSE, AxisGroupKin_Inst: AxisGroupKin_Inst)
_END_FBD_
(* the same logic as Structured Text *)
(* Network 1 *)
fbPRG_XYZ_PICKnPLACE_SFC(SFCReset := FALSE, SFCPause := FALSE, SFCTipMode := FALSE, SFCTip := FALSE, SFCEnableLimit := FALSE, SFCQuitError := FALSE, AxisGroupKin_Inst := AxisGroupKin_Inst);
END_ACTION

ACTION S350_XYZ_TARG_LIN_CIRC_ST_entry:
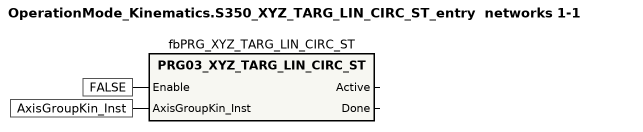
_FBD_ (* Function Block Diagram *)
NETWORK 1
	fbPRG_XYZ_TARG_LIN_CIRC_ST:PRG03_XYZ_TARG_LIN_CIRC_ST(Enable: FALSE, AxisGroupKin_Inst: AxisGroupKin_Inst)
_END_FBD_
(* the same logic as Structured Text *)
(* Network 1 *)
fbPRG_XYZ_TARG_LIN_CIRC_ST(Enable := FALSE, AxisGroupKin_Inst := AxisGroupKin_Inst);
END_ACTION

ACTION S350_XYZ_TARG_LIN_CIRC_ST_action:
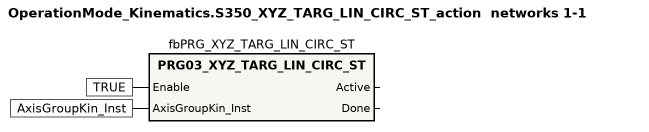
_FBD_ (* Function Block Diagram *)
NETWORK 1
	fbPRG_XYZ_TARG_LIN_CIRC_ST:PRG03_XYZ_TARG_LIN_CIRC_ST(Enable: TRUE, AxisGroupKin_Inst: AxisGroupKin_Inst)
_END_FBD_
(* the same logic as Structured Text *)
(* Network 1 *)
fbPRG_XYZ_TARG_LIN_CIRC_ST(Enable := TRUE, AxisGroupKin_Inst := AxisGroupKin_Inst);
END_ACTION

ACTION S400_XYZ_TARG_LIN_CIRC_SFC_entry:
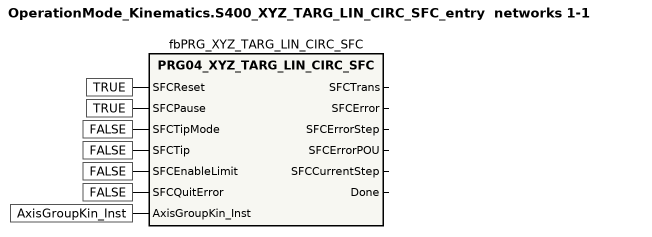
_FBD_ (* Function Block Diagram *)
NETWORK 1
	fbPRG_XYZ_TARG_LIN_CIRC_SFC:PRG04_XYZ_TARG_LIN_CIRC_SFC(SFCReset: TRUE, SFCPause: TRUE, SFCTipMode: FALSE, SFCTip: FALSE, SFCEnableLimit: FALSE, SFCQuitError: FALSE, AxisGroupKin_Inst: AxisGroupKin_Inst)
_END_FBD_
(* the same logic as Structured Text *)
(* Network 1 *)
fbPRG_XYZ_TARG_LIN_CIRC_SFC(SFCReset := TRUE, SFCPause := TRUE, SFCTipMode := FALSE, SFCTip := FALSE, SFCEnableLimit := FALSE, SFCQuitError := FALSE, AxisGroupKin_Inst := AxisGroupKin_Inst);
END_ACTION

ACTION S400_XYZ_TARG_LIN_CIRC_SFC_action:
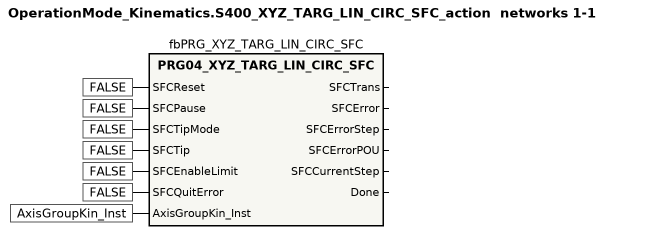
_FBD_ (* Function Block Diagram *)
NETWORK 1
	fbPRG_XYZ_TARG_LIN_CIRC_SFC:PRG04_XYZ_TARG_LIN_CIRC_SFC(SFCReset: FALSE, SFCPause: FALSE, SFCTipMode: FALSE, SFCTip: FALSE, SFCEnableLimit: FALSE, SFCQuitError: FALSE, AxisGroupKin_Inst: AxisGroupKin_Inst)
_END_FBD_
(* the same logic as Structured Text *)
(* Network 1 *)
fbPRG_XYZ_TARG_LIN_CIRC_SFC(SFCReset := FALSE, SFCPause := FALSE, SFCTipMode := FALSE, SFCTip := FALSE, SFCEnableLimit := FALSE, SFCQuitError := FALSE, AxisGroupKin_Inst := AxisGroupKin_Inst);
END_ACTION

ACTION S450_XYZ_USER_ST_entry:
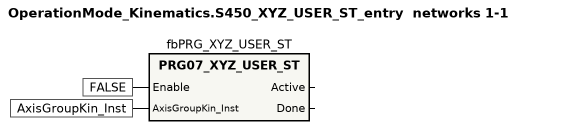
_FBD_ (* Function Block Diagram *)
NETWORK 1
	fbPRG_XYZ_USER_ST:PRG07_XYZ_USER_ST(Enable: FALSE, AxisGroupKin_Inst: AxisGroupKin_Inst)
_END_FBD_
(* the same logic as Structured Text *)
(* Network 1 *)
fbPRG_XYZ_USER_ST(Enable := FALSE, AxisGroupKin_Inst := AxisGroupKin_Inst);
END_ACTION

ACTION S450_XYZ_USER_ST_action:
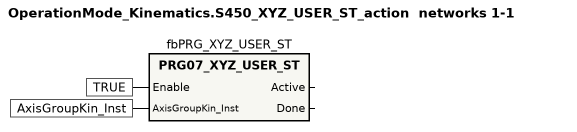
_FBD_ (* Function Block Diagram *)
NETWORK 1
	fbPRG_XYZ_USER_ST:PRG07_XYZ_USER_ST(Enable: TRUE, AxisGroupKin_Inst: AxisGroupKin_Inst)
_END_FBD_
(* the same logic as Structured Text *)
(* Network 1 *)
fbPRG_XYZ_USER_ST(Enable := TRUE, AxisGroupKin_Inst := AxisGroupKin_Inst);
END_ACTION

ACTION S500_XYZ_USER_SFC_entry:
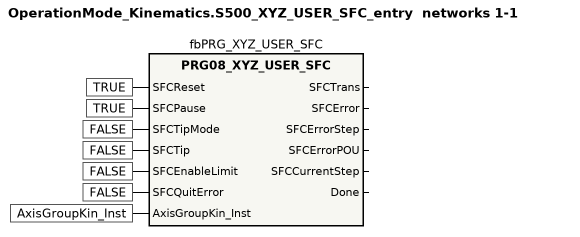
_FBD_ (* Function Block Diagram *)
NETWORK 1
	fbPRG_XYZ_USER_SFC:PRG08_XYZ_USER_SFC(SFCReset: TRUE, SFCPause: TRUE, SFCTipMode: FALSE, SFCTip: FALSE, SFCEnableLimit: FALSE, SFCQuitError: FALSE, AxisGroupKin_Inst: AxisGroupKin_Inst)
_END_FBD_
(* the same logic as Structured Text *)
(* Network 1 *)
fbPRG_XYZ_USER_SFC(SFCReset := TRUE, SFCPause := TRUE, SFCTipMode := FALSE, SFCTip := FALSE, SFCEnableLimit := FALSE, SFCQuitError := FALSE, AxisGroupKin_Inst := AxisGroupKin_Inst);
END_ACTION

ACTION S500_XYZ_USER_SFC_action:
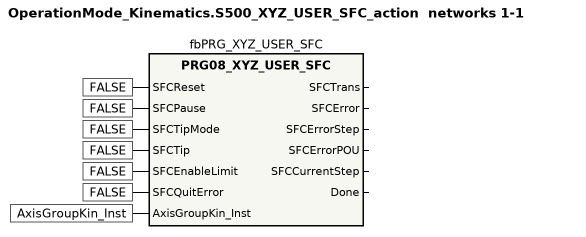
_FBD_ (* Function Block Diagram *)
NETWORK 1
	fbPRG_XYZ_USER_SFC:PRG08_XYZ_USER_SFC(SFCReset: FALSE, SFCPause: FALSE, SFCTipMode: FALSE, SFCTip: FALSE, SFCEnableLimit: FALSE, SFCQuitError: FALSE, AxisGroupKin_Inst: AxisGroupKin_Inst)
_END_FBD_
(* the same logic as Structured Text *)
(* Network 1 *)
fbPRG_XYZ_USER_SFC(SFCReset := FALSE, SFCPause := FALSE, SFCTipMode := FALSE, SFCTip := FALSE, SFCEnableLimit := FALSE, SFCQuitError := FALSE, AxisGroupKin_Inst := AxisGroupKin_Inst);
END_ACTION

ACTION S550_XYZ_FillQueue_LIN3D_with_Array_ST_entry:
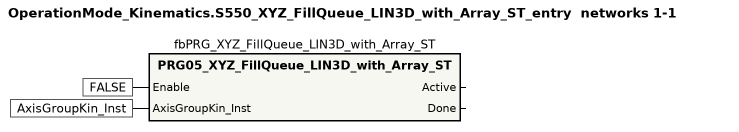
_FBD_ (* Function Block Diagram *)
NETWORK 1
	fbPRG_XYZ_FillQueue_LIN3D_with_Array_ST:PRG05_XYZ_FillQueue_LIN3D_with_Array_ST(Enable: FALSE, AxisGroupKin_Inst: AxisGroupKin_Inst)
_END_FBD_
(* the same logic as Structured Text *)
(* Network 1 *)
fbPRG_XYZ_FillQueue_LIN3D_with_Array_ST(Enable := FALSE, AxisGroupKin_Inst := AxisGroupKin_Inst);
END_ACTION

ACTION S550_XYZ_FillQueue_LIN3D_with_Array_ST_action:
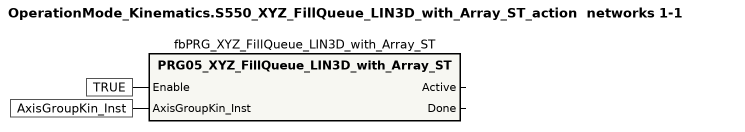
_FBD_ (* Function Block Diagram *)
NETWORK 1
	fbPRG_XYZ_FillQueue_LIN3D_with_Array_ST:PRG05_XYZ_FillQueue_LIN3D_with_Array_ST(Enable: TRUE, AxisGroupKin_Inst: AxisGroupKin_Inst)
_END_FBD_
(* the same logic as Structured Text *)
(* Network 1 *)
fbPRG_XYZ_FillQueue_LIN3D_with_Array_ST(Enable := TRUE, AxisGroupKin_Inst := AxisGroupKin_Inst);
END_ACTION

ACTION S600_XYZ_FillQueue_LIN3D_with_Array_SFC_entry:
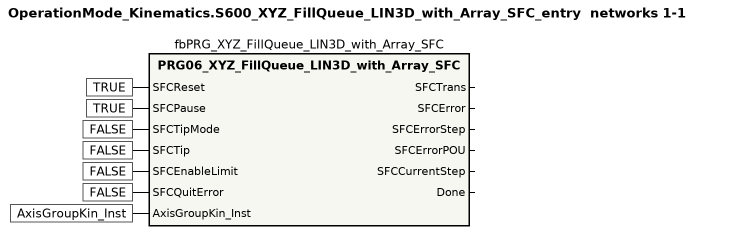
_FBD_ (* Function Block Diagram *)
NETWORK 1
	fbPRG_XYZ_FillQueue_LIN3D_with_Array_SFC:PRG06_XYZ_FillQueue_LIN3D_with_Array_SFC(SFCReset: TRUE, SFCPause: TRUE, SFCTipMode: FALSE, SFCTip: FALSE, SFCEnableLimit: FALSE, SFCQuitError: FALSE, AxisGroupKin_Inst: AxisGroupKin_Inst)
_END_FBD_
(* the same logic as Structured Text *)
(* Network 1 *)
fbPRG_XYZ_FillQueue_LIN3D_with_Array_SFC(SFCReset := TRUE, SFCPause := TRUE, SFCTipMode := FALSE, SFCTip := FALSE, SFCEnableLimit := FALSE, SFCQuitError := FALSE, AxisGroupKin_Inst := AxisGroupKin_Inst);
END_ACTION

ACTION S600_XYZ_FillQueue_LIN3D_with_Array_SFC_action:
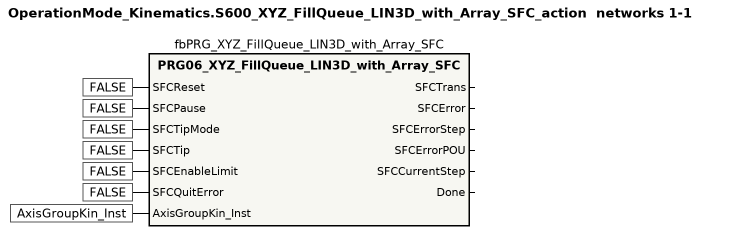
_FBD_ (* Function Block Diagram *)
NETWORK 1
	fbPRG_XYZ_FillQueue_LIN3D_with_Array_SFC:PRG06_XYZ_FillQueue_LIN3D_with_Array_SFC(SFCReset: FALSE, SFCPause: FALSE, SFCTipMode: FALSE, SFCTip: FALSE, SFCEnableLimit: FALSE, SFCQuitError: FALSE, AxisGroupKin_Inst: AxisGroupKin_Inst)
_END_FBD_
(* the same logic as Structured Text *)
(* Network 1 *)
fbPRG_XYZ_FillQueue_LIN3D_with_Array_SFC(SFCReset := FALSE, SFCPause := FALSE, SFCTipMode := FALSE, SFCTip := FALSE, SFCEnableLimit := FALSE, SFCQuitError := FALSE, AxisGroupKin_Inst := AxisGroupKin_Inst);
END_ACTION

ACTION S250_XYZ_PICKnPLACE_ST_entry:
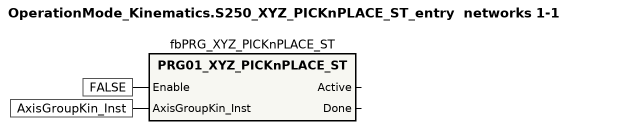
_FBD_ (* Function Block Diagram *)
NETWORK 1
	fbPRG_XYZ_PICKnPLACE_ST:PRG01_XYZ_PICKnPLACE_ST(Enable: FALSE, AxisGroupKin_Inst: AxisGroupKin_Inst)
_END_FBD_
(* the same logic as Structured Text *)
(* Network 1 *)
fbPRG_XYZ_PICKnPLACE_ST(Enable := FALSE, AxisGroupKin_Inst := AxisGroupKin_Inst);
END_ACTION

ACTION S250_XYZ_PICKnPLACE_ST_action:
